FUNCTION_BLOCK RNoAvThenRAv (* Basic Function Block Type *)
  (* Standard: 61499-2 *)
  (* Version 0.0, 8/10/2026, Schneider Electric, Template *)
  PACKAGE SE.Nereda;
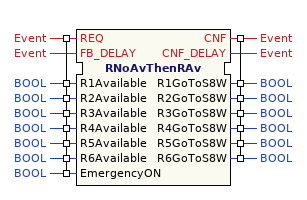
  EVENT_INPUT
    REQ WITH R1Available, R2Available, R3Available, R4Available, R5Available, R6Available, EmergencyON; (* Normal Execution Request *)
    FB_DELAY;
  END_EVENT
  EVENT_OUTPUT
    CNF WITH R1GoToS8W, R2GoToS8W, R3GoToS8W, R4GoToS8W, R5GoToS8W, R6GoToS8W; (* Execution Confirmation *)
    CNF_DELAY;
  END_EVENT
  VAR_INPUT
    R1Available : BOOL; (* Input event qualifier *)
    R2Available : BOOL;
    R3Available : BOOL;
    R4Available : BOOL;
    R5Available : BOOL;
    R6Available : BOOL;
    EmergencyON : BOOL;
  END_VAR
  VAR_OUTPUT
    R1GoToS8W : BOOL; (* Output event qualifier *)
    R2GoToS8W : BOOL;
    R3GoToS8W : BOOL;
    R4GoToS8W : BOOL;
    R5GoToS8W : BOOL;
    R6GoToS8W : BOOL;
  END_VAR
  VAR
    MemoR1Available : BOOL;
    MemoR2Available : BOOL;
    MemoR3Available : BOOL;
    MemoR4Available : BOOL;
    MemoR5Available : BOOL;
    MemoR6Available : BOOL;
  END_VAR
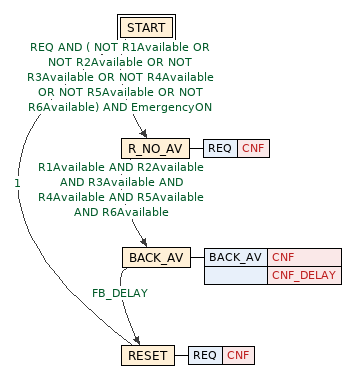
  EC_STATES
    START; (* Initial State *)
    R_NO_AV : REQ -> CNF;
    BACK_AV : BACK_AV -> CNF, -> CNF_DELAY;
    RESET : REQ -> CNF;
  END_STATES
  EC_TRANSITIONS
    START TO R_NO_AV := REQ AND ( NOT R1Available OR NOT R2Available OR NOT R3Available OR NOT R4Available OR NOT R5Available OR NOT R6Available) AND EmergencyON;
    R_NO_AV TO BACK_AV := R1Available AND R2Available AND R3Available AND R4Available AND R5Available AND R6Available;
    RESET TO START := 1;
    BACK_AV TO RESET := FB_DELAY;
  END_TRANSITIONS
  ALGORITHM REQ IN ST:
;
MemoR1Available := R1Available;
MemoR2Available := R2Available;
MemoR3Available := R3Available;
MemoR4Available := R4Available;
MemoR5Available := R5Available;
MemoR6Available := R6Available;

R1GoToS8W := FALSE;
R2GoToS8W := FALSE;
R3GoToS8W := FALSE;
R4GoToS8W := FALSE;
R5GoToS8W := FALSE;
R6GoToS8W := FALSE;
  END_ALGORITHM
  ALGORITHM BACK_AV IN ST:
;
R1GoToS8W := FALSE;
R2GoToS8W := FALSE;
R3GoToS8W := FALSE;
R4GoToS8W := FALSE;
R5GoToS8W := FALSE;
R6GoToS8W := FALSE;

IF NOT MemoR1Available THEN
    R1GoToS8W := TRUE;
END_IF;

IF NOT MemoR2Available THEN
    R2GoToS8W := TRUE;
END_IF;

IF NOT MemoR3Available THEN
    R3GoToS8W := TRUE;
END_IF;

IF NOT MemoR4Available THEN
    R4GoToS8W := TRUE;
END_IF;

IF NOT MemoR5Available THEN
    R5GoToS8W := TRUE;
END_IF;

IF NOT MemoR6Available THEN
    R6GoToS8W := TRUE;
END_IF;
  END_ALGORITHM
END_FUNCTION_BLOCK
